// TIA Portal V17 export
// export: Created 2025-06-26T06:49:22.3940312Z, ExportSetting WithDefaults, DisplayName Totally Integrated Automation Portal, DisplayVersion V17 Update 8, DisplayName TIA Portal Openness, DisplayVersion V17 Update 8, DisplayName TIA Portal Version Control Interface, DisplayVersion V17, DisplayName STEP 7 Professional, DisplayVersion V17 Update 8, DisplayName STEP 7 Safety, DisplayVersion V17 Update 6, DisplayName WinCC Advanced, DisplayVersion V17 Update 8
DATA_BLOCK "DB_Customer"   // DB10
{ S7_Optimized_Access := 'TRUE' }
AUTHOR : Heaten
VERSION : 0.1
// stored: AutoNumber true, DBAccessibleFromOPCUA true, IsOnlyStoredInLoadMemory false, IsRetainMemResEnabled false, IsWriteProtectedInAS false, MemoryReserve 100
   VAR
      bEnabled : Bool;   // Enable Customer interface
      Watchdog : "stHeartbeatCount2";   // Comm monitoring Customer <-> Heatbooster
      Dummy { S7_SetPoint := 'True'} : "stCalcValue";
   END_VAR
BEGIN
END_DATA_BLOCK
